FUNCTION_BLOCK sequence_Pattern_04_04_loop_AX (* Pattern Sequence 4 Steps 4 Outputs (Cam Sequencer), AX Adapter *)
  (* Standard: 61499-2; Description: Copyright (c) 2026 HR Agrartechnik GmbH This program and the accompanying materials are made available under the terms of the Eclipse Public License 2.0 which is available at https://www.eclipse.org/legal/epl-2.0/ SPDX-License-Identifier: EPL-2.0 *)
  (* Version 1.0, 2026-02-01, Franz Höpfinger, HR Agrartechnik GmbH *)
  PACKAGE logiBUS::utils::sequence::pattern;
  IMPORT logiBUS::utils::sequence::const::sequence;
  IMPORT logiBUS::utils::sequence::const::sequence::NO_TIME;
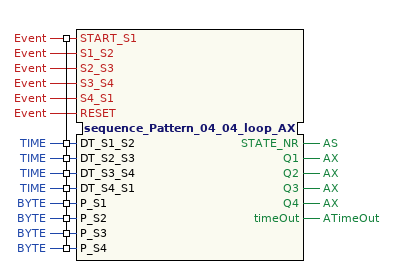
  EVENT_INPUT
    START_S1 WITH DT_S1_S2, DT_S2_S3, DT_S3_S4, DT_S4_S1, P_S1, P_S2, P_S3, P_S4; (* jump from START to State_01 *)
    S1_S2; (* jump from State_01 to State_02 *)
    S2_S3; (* jump from State_02 to State_03 *)
    S3_S4; (* jump from State_03 to State_04 *)
    S4_S1; (* jump from State_04 to State_01 *)
    RESET; (* Reset from any State to START *)
  END_EVENT
  VAR_INPUT
    DT_S1_S2 : TIME := NO_TIME; (* State_01 to State_02 timed *)
    DT_S2_S3 : TIME := NO_TIME; (* State_02 to State_03 timed *)
    DT_S3_S4 : TIME := NO_TIME; (* State_03 to State_04 timed *)
    DT_S4_S1 : TIME := NO_TIME; (* State_04 to State_01 timed *)
    P_S1 : BYTE := 1; (* Pattern for State 01 (Bit0=Q1, Bit1=Q2...) *)
    P_S2 : BYTE := 2; (* Pattern for State 02 *)
    P_S3 : BYTE := 4; (* Pattern for State 03 *)
    P_S4 : BYTE := 8; (* Pattern for State 04 *)
  END_VAR
  PLUGS
    STATE_NR : adapter::types::unidirectional::AS; (* State Number Adapter *)
    Q1 : adapter::types::unidirectional::AX; (* Output 1 (Bit 0) *)
    Q2 : adapter::types::unidirectional::AX; (* Output 2 (Bit 1) *)
    Q3 : adapter::types::unidirectional::AX; (* Output 3 (Bit 2) *)
    Q4 : adapter::types::unidirectional::AX; (* Output 4 (Bit 3) *)
    timeOut : iec61499::events::ATimeOut; (* timeOut Adapter *)
  END_PLUGS
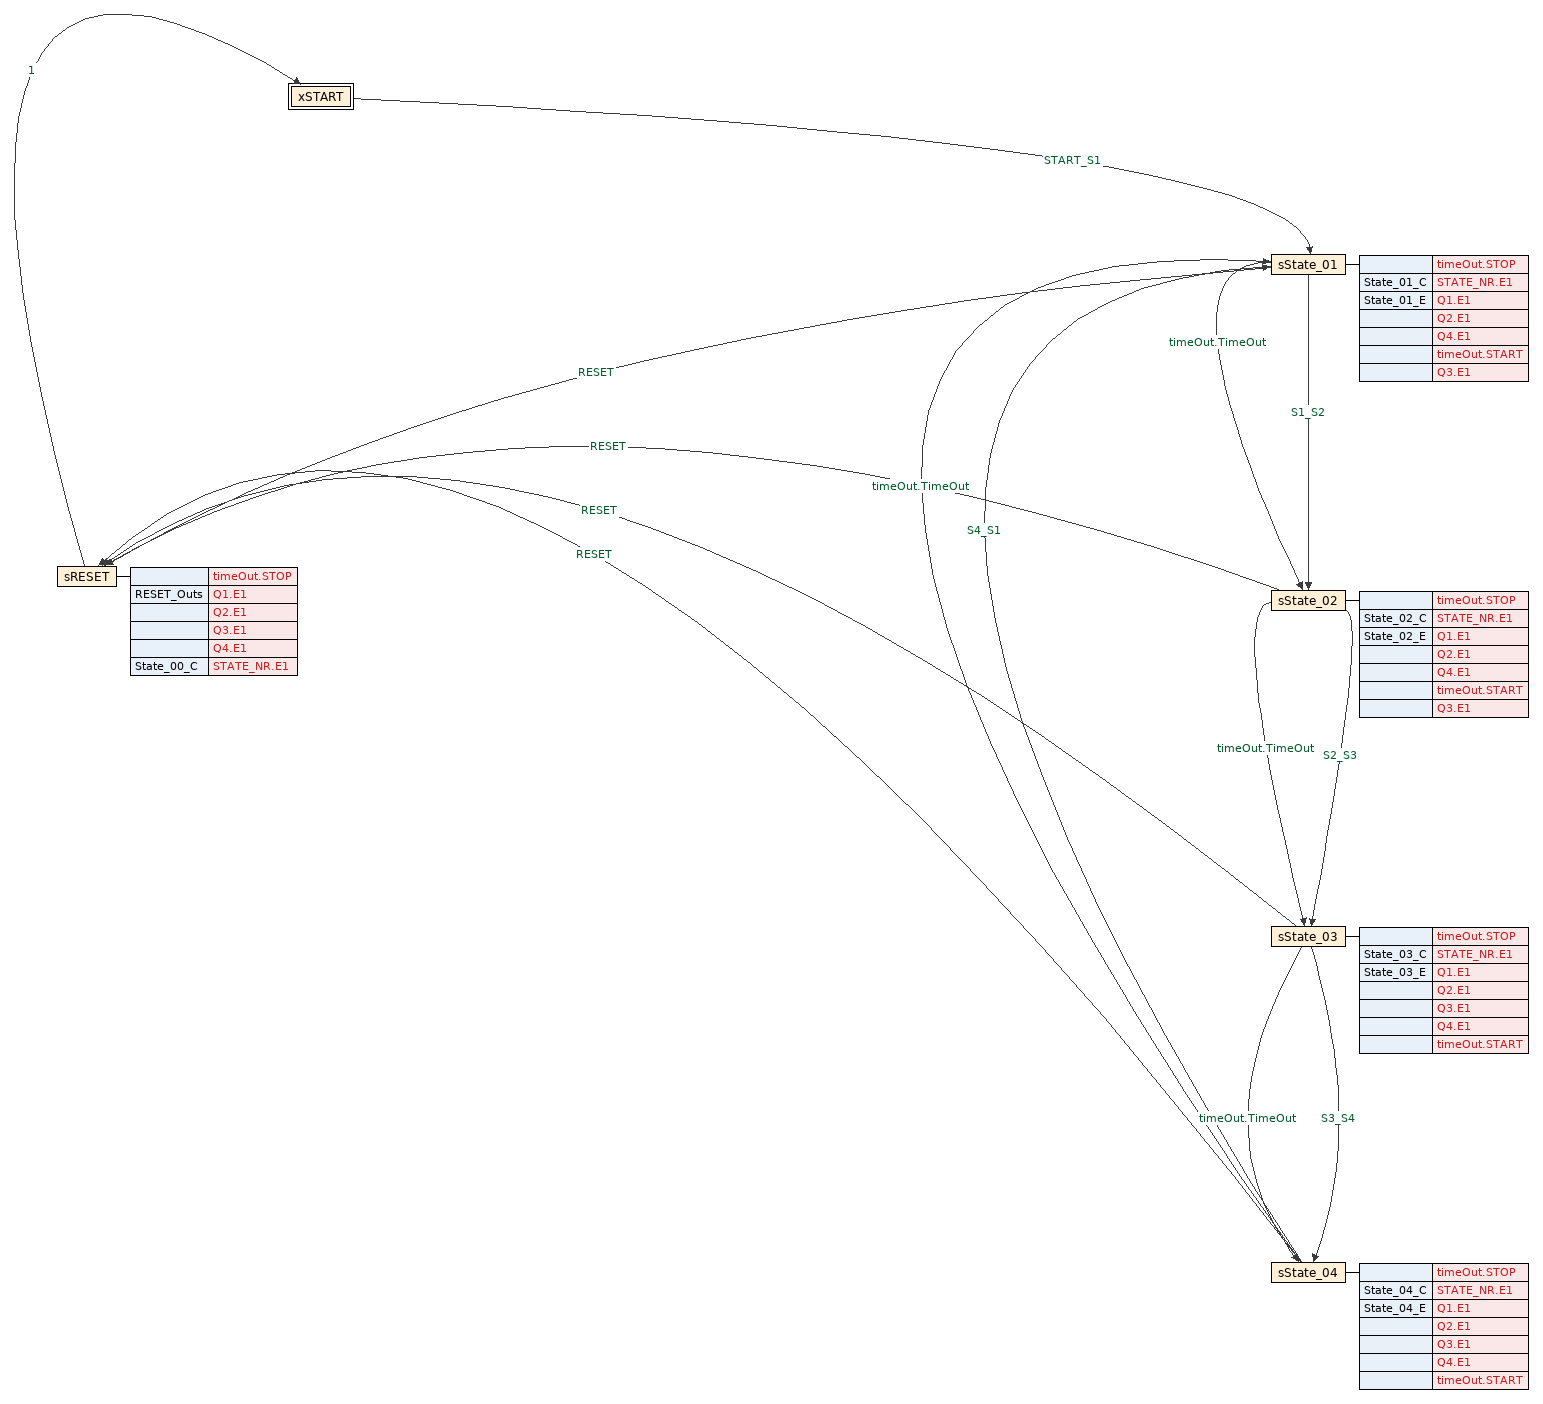
  EC_STATES
    xSTART; (* Initial State *)
    sState_01 : -> timeOut.STOP, State_01_C -> STATE_NR.E1, State_01_E -> Q1.E1, -> Q2.E1, -> Q4.E1, -> timeOut.START, -> Q3.E1;
    sState_02 : -> timeOut.STOP, State_02_C -> STATE_NR.E1, State_02_E -> Q1.E1, -> Q2.E1, -> Q4.E1, -> timeOut.START, -> Q3.E1;
    sState_03 : -> timeOut.STOP, State_03_C -> STATE_NR.E1, State_03_E -> Q1.E1, -> Q2.E1, -> Q3.E1, -> Q4.E1, -> timeOut.START;
    sState_04 : -> timeOut.STOP, State_04_C -> STATE_NR.E1, State_04_E -> Q1.E1, -> Q2.E1, -> Q3.E1, -> Q4.E1, -> timeOut.START;
    sRESET : -> timeOut.STOP, RESET_Outs -> Q1.E1, -> Q2.E1, -> Q3.E1, -> Q4.E1, State_00_C -> STATE_NR.E1;
  END_STATES
  EC_TRANSITIONS
    sState_01 TO sState_02 := S1_S2;
    sState_02 TO sState_03 := S2_S3;
    sState_03 TO sState_04 := S3_S4;
    sState_01 TO sState_02 := timeOut.TimeOut;
    sState_02 TO sState_03 := timeOut.TimeOut;
    sState_03 TO sState_04 := timeOut.TimeOut;
    xSTART TO sState_01 := START_S1;
    sState_01 TO sRESET := RESET;
    sState_04 TO sRESET := RESET;
    sState_02 TO sRESET := RESET;
    sState_03 TO sRESET := RESET;
    sState_04 TO sState_01 := S4_S1;
    sState_04 TO sState_01 := timeOut.TimeOut;
    sRESET TO xSTART := 1;
  END_TRANSITIONS
  ALGORITHM State_00_C IN ST:
STATE_NR.D1 := sequence::State_00;
  END_ALGORITHM
  ALGORITHM State_01_C IN ST:
STATE_NR.D1 := sequence::State_01;
timeOut.DT := DT_S1_S2;
  END_ALGORITHM
  ALGORITHM State_02_C IN ST:
STATE_NR.D1 := sequence::State_02;
timeOut.DT := DT_S2_S3;
  END_ALGORITHM
  ALGORITHM State_03_C IN ST:
STATE_NR.D1 := sequence::State_03;
timeOut.DT := DT_S3_S4;
  END_ALGORITHM
  ALGORITHM State_04_C IN ST:
STATE_NR.D1 := sequence::State_04;
timeOut.DT := DT_S4_S1;
  END_ALGORITHM
  ALGORITHM State_01_E IN ST:
Q1.D1 := P_S1.0;
Q2.D1 := P_S1.1;
Q3.D1 := P_S1.2;
Q4.D1 := P_S1.3;
  END_ALGORITHM
  ALGORITHM State_02_E IN ST:
Q1.D1 := P_S2.0;
Q2.D1 := P_S2.1;
Q3.D1 := P_S2.2;
Q4.D1 := P_S2.3;
  END_ALGORITHM
  ALGORITHM State_03_E IN ST:
Q1.D1 := P_S3.0;
Q2.D1 := P_S3.1;
Q3.D1 := P_S3.2;
Q4.D1 := P_S3.3;
  END_ALGORITHM
  ALGORITHM State_04_E IN ST:
Q1.D1 := P_S4.0;
Q2.D1 := P_S4.1;
Q3.D1 := P_S4.2;
Q4.D1 := P_S4.3;
  END_ALGORITHM
  ALGORITHM RESET_Outs IN ST:
Q1.D1 := FALSE;
Q2.D1 := FALSE;
Q3.D1 := FALSE;
Q4.D1 := FALSE;
  END_ALGORITHM
END_FUNCTION_BLOCK
